PROGRAM MAIN
VAR_INPUT
	enable : BOOL;
	reset : BOOL;
	
	positive : BOOL;
	negative : BOOL;
	
	target : LREAL := 1;
END_VAR
VAR
	servo : ServoNC;
END_VAR

servo(
	bEnable:= enable, 
	home=> , 
	outerLimit=> , 
	innerLimit=> , 
	ready=> , 
	busy=> , 
	error=> , 
	homeSet=> , 
	position=> );

IF NOT servo.homeSet THEN
	servo.homingSequence();
	RETURN;
END_IF

servo.stop();

IF positive THEN
	servo.moveContinuous(direction:= MC_Positive_Direction);
	negative := FALSE;
END_IF

IF negative THEN
	servo.moveContinuous(direction:= MC_Negative_Direction);
	positive := FALSE;
END_IF

IF target < 0 THEN
	servo.moveAbsolute(target);
END_IF

IF reset THEN
	servo.reset();
	reset := FALSE;
END_IF

END_PROGRAM

(* stored: Version 1.1.0.1, ProductVersion 3.1.4024.11
   POU MAIN: Id {1f5f61ca-3148-4cc9-a992-52c18d091d4f}, SpecialFunc None *)
